// TIA Portal V18 export
DATA_BLOCK "LoadCell_FluidTankWeight_DB"   // DB23
VERSION : 0.1
// stored: AutoNumber true, DBAccessibleFromOPCUA true, InstanceOfName LoadCell, InstanceOfType FB
"LoadCell"
   // VAR_INPUT
   //    MinValue : UInt;
   //    MaxValue : UInt;
   //    ILoadCell : UInt;
   //    Const_V : UInt;
   //    Const_SubWeight : Real;
   //    Const_Kg : UInt;
   // END_VAR
   // VAR_OUTPUT
   //    OWeight : UInt;
   // END_VAR
BEGIN
END_DATA_BLOCK
